Fanuc KAREL source: kb00018.KL

PROGRAM KB00018
%NOLOCKGROUP
VAR
P1 : XYZWPREXT;P2 : POSITION;P3 : POSITION;P4:INTEGER
BEGIN
--
--
--
P4=1
CHECK_EPOS(P1,P2,P3,P4,1)
END KB00018
